// TIA Portal V20 export
DATA_BLOCK "PRODDATA_HMI_IF_DB"   // DB30439
TITLE = HMI und Anwender Schnittstelle für Produktionsdaten / HMI and user interface for production data
{ S7_Optimized_Access := 'TRUE' }
AUTHOR : SICAR
FAMILY : ProdData
// FUNKTIONSBESCHREIBUNG: 
// Der Baustein beinhaltet alle Informationen zum und vom HMI, sowie die Anwenderschnittstellen für die Produktionsdaten
// Weitere Hinweise: siehe SICAR anwenderdefinierte Dokumentation / SICAR Online-Hilfe.
// DESCRIPTION OF FUNCTIONS:
// stored: AutoNumber false, MemoryReserve 100
   VAR
      No_DataSets : Struct   // Anzahl konfigurierter Datensätze / Information number of DataSets
         Limits : Int;
         "Timer" : Int;
         "Counter" : Int;
         ShiftCounter : Int;
      END_STRUCT;
      Limit_ColorCode_Summary : UInt;
      Limit_ColorCode_SelectButton : Array[0..8] of UInt;   // Farbcode für Datensatz Anwahl Button (Grenzwerte) / Color code for data-set select button (Limit values)
   END_VAR
   VAR RETAIN
      Limit_DataSet { S7_SetPoint := 'True'} : Array[0.."No_of_DataSets_LimitValues"] of "LIMIT_VALUE_UDT_1";   // Datensätze Grenzwerte / DataSets Limit value
      CycleTimer_DataSet { S7_SetPoint := 'True'} : Array[0.."No_of_DataSets_CycleTimer"] of "CYCLE_TIMER_UDT";   // Datensätze Taktzeiten / DataSets Cycle timer
      Counter_DataSet { S7_SetPoint := 'True'} : Array[0.."No_of_DataSets_Counter"] of "COUNTER_UDT";   // Datensätze Zähler
      ShiftCounter_DataSet { S7_SetPoint := 'True'} : Array[0.."No_of_DataSets_ShiftCounter"] of "SHIFT_COUNTER_UDT";   // Datensätze Schichtzähler / DataSets ShiftCounter
      "ShiftCounter+OEE+TREND_DataSet" { S7_SetPoint := 'True'} : Array[0.."No_of_DataSets_ShiftCounter"] of "SHIFT_COUNTER_OEE_TREND_UDT";   // Datensätze Schichtzähler / DataSets ShiftCounter
   END_VAR
BEGIN
END_DATA_BLOCK
